FUNCTION_BLOCK Fb_SystemVariables
VAR
	// **** Function blocks *****
		Fb_SystemTime: FB_LocalSystemTime ;
		Fb_TimerHbOn : Ton ; // Timer Heartbeat on
		Fb_TimerFast : Ton ; // Timer for fast blink bit
		Fb_TimerSlow : Ton ; // Timer for slow blink bit
		Fb_RisingPulse : R_Trig ; // Rinsing edge trigger function	
	// ***** internal Variables *****
		HeartbeatOn	: BOOL ; // heartbeat is on
		FlashFastOn	: BOOL ; // Fast Flash bit on
		FlashSlowOn	: BOOL ; // Flash slow bit on
	
		Fb_Timer100mSec : TON := (PT := T#100MS); // Timer for 100 ms pulse
		
		fbFormatString : FB_FormatString;
END_VAR

// ===== Get system time =====
	// ***** get windows system time *****
		Fb_SystemTime(	sNetID := '', 
						bEnable := TRUE, 
						dwCycle := 1,
						dwOpt := 0, 
						tTimeout := DEFAULT_ADS_TIMEOUT, 	
						systemTime => Sys_Variables.SystemTime_TS,
						tzID	=> Sys_Variables.TimeZoneId
						);
	// ****** convert to time of day format *****
		Sys_Variables.SystemTime := SYSTEMTIME_TO_DT(TIMESTR := Sys_Variables.SystemTime_TS) ;
		
	// Create a timestamp string
	Sys_Variables.SystemTimeString := CreateTimestampString();

// ===== Heartbeat generator =====
	Fb_TimerHbOn(In := NOT HeartbeatOn , PT:= T#1S, Q => HeartbeatOn);
	IF Fb_TimerHbOn.ET >= T#500MS THEN
		Sys_Variables.HeartBeat := TRUE ;
	ELSE
		Sys_Variables.HeartBeat := FALSE ;
	END_IF

// ===== one second pulse generator =====
	Fb_RisingPulse(Clk := HeartbeatOn, Q => Sys_Variables.Pulse1Sec);
	
// ===== 100ms pulse generation ======
	Fb_Timer100mSec( IN := NOT Sys_Variables.Pulse100ms, Q => Sys_Variables.Pulse100ms);

// ===== Flash fast bit =====
	Fb_TimerFast(In := NOT FlashFastOn, Pt := T#1S, Q => FlashFastOn);
	IF Fb_TimerFast.ET >= T#600MS THEN
		Sys_Variables.BlinkFast := TRUE;  
	ELSE
		Sys_Variables.BlinkFast := FALSE;  		
	END_IF
// ===== Flash Slow bit =====
	Fb_TimerSlow(In := NOT FlashSLowOn, Pt := T#2S, Q => FlashSlowOn);
	IF Fb_TimerSlow.ET >= T#1200MS THEN
		Sys_Variables.BlinkSlow := TRUE;  
	ELSE
		Sys_Variables.BlinkSlow := FALSE;  		
	END_IF

// ===== Always true and always false bits =====
	Sys_Variables.AlwaysOff := FALSE 	;
	Sys_Variables.AlwaysOn	:= TRUE		;
	
// ===== Manage persistent data ======
	DataManager.FbPersistentManager();

METHOD PROTECTED CreateTimestampString : STRING[21]
VAR
	fMonth : REAL;
	fDay : REAL;
	fHour : REAL;
	fMinute : REAL;
	fSecond : REAL;
	fMilliseconds : REAL;
END_VAR
// Suppress error "VAR_IN_OUT parameter 'in' needs variable with write access as input."	
fMonth := WORD_TO_REAL(Sys_Variables.SystemTime_TS.wMonth); 
fDay := WORD_TO_REAL(Sys_Variables.SystemTime_TS.wDay); 
fHour := WORD_TO_REAL(Sys_Variables.SystemTime_TS.wHour); 
fMinute := WORD_TO_REAL(Sys_Variables.SystemTime_TS.wMinute); 
fSecond := WORD_TO_REAL(Sys_Variables.SystemTime_TS.wSecond); 
fMilliseconds := WORD_TO_REAL(Sys_Variables.SystemTime_TS.wMilliseconds); 

fbFormatString(
	sFormat := '%u%02.0f%02.0f-%02.0f:%02.0f:%02.0f.%03.0f',
	arg1 := F_WORD(Sys_Variables.SystemTime_TS.wYear),
	arg2 := F_REAL(fMonth),
	arg3 := F_REAL(fDay),
	arg4 := F_REAL(fHour),
	arg5 := F_REAL(fMinute),
	arg6 := F_REAL(fSecond),
	arg7 := F_REAL(fMilliseconds),
	sOut => CreateTimestampString
);
END_METHOD

END_FUNCTION_BLOCK

(* stored: Version 1.1.0.1, ProductVersion 3.1.4024.11
   POU Fb_SystemVariables: Id {da83f45a-6f6a-41cc-bbb4-a67342500421}, SpecialFunc None
   Method CreateTimestampString: Id {7fc4e248-6970-0169-32d9-f97ed5a3eae6} *)
